{attribute addProperty BoxType "EK1122-0000-0018"}
{attribute addProperty Id "Beckhoff_EPP3xxxsub_EK1100EK1100_179A0949162A_0001_EPP3174_0002_0016EPP3174_83515A0D22428A_0002_EPP3174_0002_0017EPP3174_83515A0D22428A_0003_EPP3174_0002_0018EPP3174_83515A0D22428A_0004_EPP3184_0002_0016EPP3184_55F04E9922428A_0005_EPP3184_0002_0017EPP3184_55F04E9922428A_0006_EPP3184_0002_0018EPP3184_55F04E9922428A_0007_EPP3184_0002_0019EPP3184_83515A0D22428A_0008_EPP3204_0002_0016EPP3204_BF093E1239249A_0009_EPP3204_0002_0017EPP3204_69AA4F8E22428A_0010_EPP3204_0002_0018EPP3204_69AA4F8E22428A_0011_EPP3204_0002_0019EPP3204_69AA4F8E22428A_0012_EPP3314_0002_0016EPP3314_2E54E3B022428A_0013_EPP3314_0002_0017EPP3314_2E54E3B022428A_0014_EPP3314_0002_0018EPP3314_2E54E3B022428A_0015_EPP3632_0001_0016EPP3632_C340233D59274A_0016_EPP3632_0001_0017EPP3632_C340233D59274A_0017_EPP3744_0041_0016EPP3744_38AF8BFB40050A_0018_EPP3744_0041_0017EPP3744_38AF8BFB40050A_0019_EPP3744_0041_0018EPP3744_38AF8BFB40050A_0020_EPP3744_1041_0016EPP3744_38AF8BFB40050A_0021_EPP3744_1041_0017EPP3744_38AF8BFB40050A_0022_EPP3744_1041_0018EPP3744_38AF8BFB40050A_0023_EPP3744_1041_0019EPP3744_38AF8BFB40050A_0024_EPP3744_1041_0020EPP3744_38AF8BFB40050A_0025_EPP3752_0000_0017EPP3752_AEF24F9C28836"}
{attribute addProperty CRC "2764646260"}
{attribute addProperty SizeInBites "7992"}
{attribute addProperty SizeInBytes "999"}
TYPE Beckhoff_EPP3xxxEK1122_A4C92774 EXTENDS EK1122_179A0949 :
STRUCT
	{attribute addProperty Name "Beckhoff_EPP3xxxsub_EK1100"}
	Beckhoff_EPP3xxxsub_EK1100 : EK1100_179A0949;
	{attribute addProperty Name "A_0001_EPP3174_0002_0016"}
	A_0001_EPP3174_0002_0016 : EPP3174_83515A0D;
	{attribute addProperty Name "A_0002_EPP3174_0002_0017"}
	A_0002_EPP3174_0002_0017 : EPP3174_83515A0D;
	{attribute addProperty Name "A_0003_EPP3174_0002_0018"}
	A_0003_EPP3174_0002_0018 : EPP3174_83515A0D;
	{attribute addProperty Name "A_0004_EPP3184_0002_0016"}
	A_0004_EPP3184_0002_0016 : EPP3184_55F04E99;
	{attribute addProperty Name "A_0005_EPP3184_0002_0017"}
	A_0005_EPP3184_0002_0017 : EPP3184_55F04E99;
	{attribute addProperty Name "A_0006_EPP3184_0002_0018"}
	A_0006_EPP3184_0002_0018 : EPP3184_55F04E99;
	{attribute addProperty Name "A_0007_EPP3184_0002_0019"}
	A_0007_EPP3184_0002_0019 : EPP3184_83515A0D;
	{attribute addProperty Name "A_0008_EPP3204_0002_0016"}
	A_0008_EPP3204_0002_0016 : EPP3204_BF093E12;
	{attribute addProperty Name "A_0009_EPP3204_0002_0017"}
	A_0009_EPP3204_0002_0017 : EPP3204_69AA4F8E;
	{attribute addProperty Name "A_0010_EPP3204_0002_0018"}
	A_0010_EPP3204_0002_0018 : EPP3204_69AA4F8E;
	{attribute addProperty Name "A_0011_EPP3204_0002_0019"}
	A_0011_EPP3204_0002_0019 : EPP3204_69AA4F8E;
	{attribute addProperty Name "A_0012_EPP3314_0002_0016"}
	A_0012_EPP3314_0002_0016 : EPP3314_2E54E3B0;
	{attribute addProperty Name "A_0013_EPP3314_0002_0017"}
	A_0013_EPP3314_0002_0017 : EPP3314_2E54E3B0;
	{attribute addProperty Name "A_0014_EPP3314_0002_0018"}
	A_0014_EPP3314_0002_0018 : EPP3314_2E54E3B0;
	{attribute addProperty Name "A_0015_EPP3632_0001_0016"}
	A_0015_EPP3632_0001_0016 : EPP3632_C340233D;
	{attribute addProperty Name "A_0016_EPP3632_0001_0017"}
	A_0016_EPP3632_0001_0017 : EPP3632_C340233D;
	{attribute addProperty Name "A_0017_EPP3744_0041_0016"}
	A_0017_EPP3744_0041_0016 : EPP3744_38AF8BFB;
	{attribute addProperty Name "A_0018_EPP3744_0041_0017"}
	A_0018_EPP3744_0041_0017 : EPP3744_38AF8BFB;
	{attribute addProperty Name "A_0019_EPP3744_0041_0018"}
	A_0019_EPP3744_0041_0018 : EPP3744_38AF8BFB;
	{attribute addProperty Name "A_0020_EPP3744_1041_0016"}
	A_0020_EPP3744_1041_0016 : EPP3744_38AF8BFB;
	{attribute addProperty Name "A_0021_EPP3744_1041_0017"}
	A_0021_EPP3744_1041_0017 : EPP3744_38AF8BFB;
	{attribute addProperty Name "A_0022_EPP3744_1041_0018"}
	A_0022_EPP3744_1041_0018 : EPP3744_38AF8BFB;
	{attribute addProperty Name "A_0023_EPP3744_1041_0019"}
	A_0023_EPP3744_1041_0019 : EPP3744_38AF8BFB;
	{attribute addProperty Name "A_0024_EPP3744_1041_0020"}
	A_0024_EPP3744_1041_0020 : EPP3744_38AF8BFB;
	{attribute addProperty Name "A_0025_EPP3752_0000_0017"}
	A_0025_EPP3752_0000_0017 : EPP3752_AEF24F9C;
END_STRUCT
END_TYPE

(* stored: Version 1.2.0.0, ProductVersion 3.1.4024.9
   DUT Beckhoff_EPP3xxxEK1122_A4C92774: Id {0299f430-137e-4efd-90fb-a266ef40adee} *)
